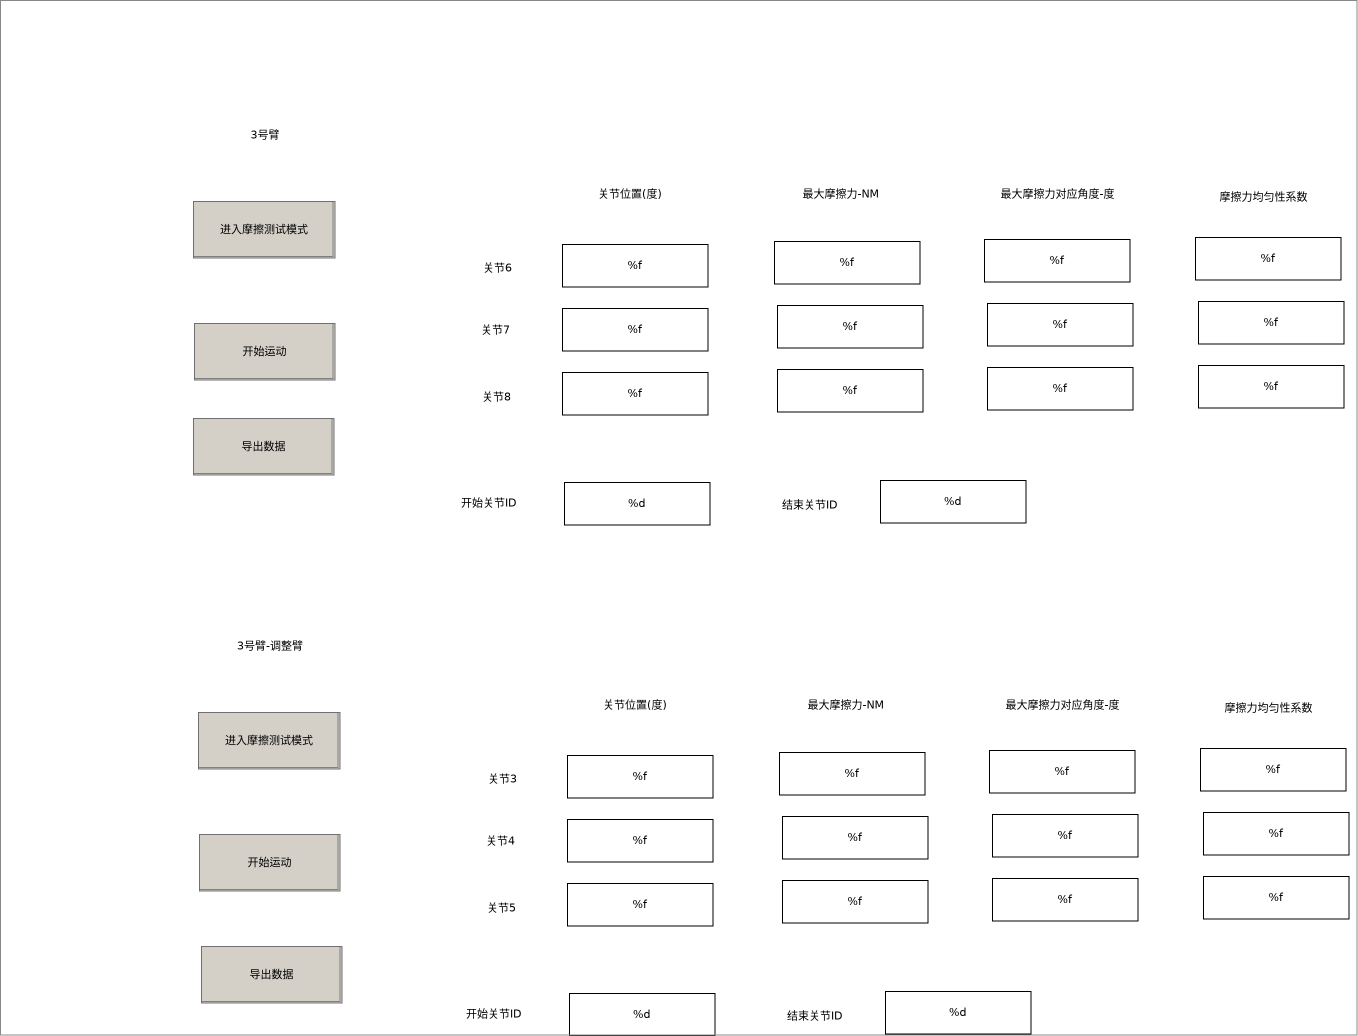
VISUALIZATION friction_a3  // 1358x1036
    Button (193,201 142x57), "进入摩擦测试模式", colour toggle: g_frictionTest.m_testMode[3]
        toggle g_frictionTest.m_testMode[3]
    Button (194,323 141x57), "开始运动", colour toggle: g_frictionTest.m_startMotion[3]
        toggle g_frictionTest.m_startMotion[3]
    Label (190,120 150x30), "3号臂"
    Rectangle (774,241 146x43), "%f", text variable: g_frictionTest.m_CoulombFrictionMax[3][1]
    Rectangle (777,305 146x43), "%f", text variable: g_frictionTest.m_CoulombFrictionMax[3][2]
    Rectangle (777,369 146x43), "%f", text variable: g_frictionTest.m_CoulombFrictionMax[3][3]
    Label (766,179 150x30), "最大摩擦力-NM"
    Rectangle (984,239 146x43), "%f", text variable: g_frictionTest.m_CoulombFrictionMax_JntPos[3][1]
    Rectangle (987,303 146x43), "%f", text variable: g_frictionTest.m_CoulombFrictionMax_JntPos[3][2]
    Rectangle (987,367 146x43), "%f", text variable: g_frictionTest.m_CoulombFrictionMax_JntPos[3][3]
    Label (941,179 233x30), "最大摩擦力对应角度-度"
    Rectangle (1195,237 146x43), "%f", text variable: g_frictionTest.m_CoulombFrictionRatio[3,1]
    Rectangle (1198,301 146x43), "%f", text variable: g_frictionTest.m_CoulombFrictionRatio[3,2]
    Rectangle (1198,365 146x43), "%f", text variable: g_frictionTest.m_CoulombFrictionRatio[3,3]
    Label (1174,182 179x30), "摩擦力均匀性系数"
    Rectangle (562,244 146x43), "%f", text variable: g_frictionTest.m_armDHJntPos[3][1]
    Label (446,250 103x36), "关节6"
    Label (444,312 103x36), "关节7"
    Label (445,379 103x36), "关节8"
    Rectangle (562,308 146x43), "%f", text variable: g_frictionTest.m_armDHJntPos[3][2]
    Rectangle (562,372 146x43), "%f", text variable: g_frictionTest.m_armDHJntPos[3][3]
    Label (555,179 150x30), "关节位置(度)"
    Label (414,488 150x30), "开始关节ID"
    Rectangle (564,482 146x43), "%d", text variable: g_frictionTest.m_jntIdStart[3]
        OnMouseClick: write the text variable via Default
    Label (735,490 150x30), "结束关节ID"
    Rectangle (880,480 146x43), "%d", text variable: g_frictionTest.m_jntIdEnd[3]
        OnMouseClick: write the text variable via Default
    Button (198,712 142x57), "进入摩擦测试模式", colour toggle: g_frictionTestSetup.m_testMode[3]
        toggle g_frictionTestSetup.m_testMode[3]
    Button (199,834 141x57), "开始运动", colour toggle: g_frictionTestSetup.m_startMotion[3]
        toggle g_frictionTestSetup.m_startMotion[3]
    Label (195,631 150x30), "3号臂-调整臂"
    Rectangle (779,752 146x43), "%f", text variable: g_frictionTestSetup.m_CoulombFrictionMax[3][3]
    Rectangle (782,816 146x43), "%f", text variable: g_frictionTestSetup.m_CoulombFrictionMax[3][4]
    Rectangle (782,880 146x43), "%f", text variable: g_frictionTestSetup.m_CoulombFrictionMax[3][5]
    Label (771,690 150x30), "最大摩擦力-NM"
    Rectangle (989,750 146x43), "%f", text variable: g_frictionTestSetup.m_CoulombFrictionMax_JntPos[3][3]
    Rectangle (992,814 146x43), "%f", text variable: g_frictionTestSetup.m_CoulombFrictionMax_JntPos[3][4]
    Rectangle (992,878 146x43), "%f", text variable: g_frictionTestSetup.m_CoulombFrictionMax_JntPos[3][5]
    Label (946,690 233x30), "最大摩擦力对应角度-度"
    Rectangle (1200,748 146x43), "%f", text variable: g_frictionTestSetup.m_CoulombFrictionRatio[3,3]
    Rectangle (1203,812 146x43), "%f", text variable: g_frictionTestSetup.m_CoulombFrictionRatio[3,4]
    Rectangle (1203,876 146x43), "%f", text variable: g_frictionTestSetup.m_CoulombFrictionRatio[3,5]
    Label (1179,693 179x30), "摩擦力均匀性系数"
    Rectangle (567,755 146x43), "%f", text variable: g_frictionTestSetup.m_armDHJntPos[3][3]
    Label (451,761 103x36), "关节3"
    Label (449,823 103x36), "关节4"
    Label (450,890 103x36), "关节5"
    Rectangle (567,819 146x43), "%f", text variable: g_frictionTestSetup.m_armDHJntPos[3][4]
    Rectangle (567,883 146x43), "%f", text variable: g_frictionTestSetup.m_armDHJntPos[3][5]
    Label (560,690 150x30), "关节位置(度)"
    Label (419,999 150x30), "开始关节ID"
    Rectangle (569,993 146x43), "%d", text variable: g_frictionTestSetup.m_jntIdStart[3]
        OnMouseClick: write the text variable via Default
    Label (740,1001 150x30), "结束关节ID"
    Rectangle (885,991 146x43), "%d", text variable: g_frictionTestSetup.m_jntIdEnd[3]
        OnMouseClick: write the text variable via Default
    Button (193,418 141x57), "导出数据", colour toggle: g_frictionTest.m_duringWriteData[3]
        tap g_frictionTest.m_writeData[3]
    Button (201,946 141x57), "导出数据", colour toggle: g_frictionTestSetup.m_duringWriteData[3]
        tap g_frictionTestSetup.m_writeData[3]
END_VISUALIZATION

(* stored: Version 1.1.0.1, ProductVersion 3.1.4024.12
   Visu friction_a3: Id {1ceb5afc-9819-4bbd-8e03-1c24eeca4f13} *)
